(*

short summary
=================
Class provides assert statements
for 8-bit windows-1252 and UTF-16 strings with an undifined length.

.. attention:: 
	All strings are handled as null terminated byte/word streams.
	For windows-1252 is end of the string 16#00
	For UTF-16 is end of the string 16#00_00

.. attention:: 
	The interface :ref:`IAnyStringAssertions` uses ``ANY_STRING``, 
	for this it's not possible to use literals/constants,
	because for ``ANY`` types generates the compiler ``__SYSTEM.AnyType``
	and ``__SYSTEM.AnyType`` contains a pointer  

.. <legal notes>

legal notes
=================
| SPDX-FileCopyrightText: © 2022 ekvip automation GmbH <info@ekvip.de>
| SPDX-License-Identifier: Apache-2.0
| For details check: Apache-2.0_

.. _Apache-2.0: https://www.apache.org/licenses/LICENSE-2.0

.. </legal notes>

methods and properties
=======================

*)

{attribute 'reflection'}
FUNCTION_BLOCK INTERNAL AnyStringAssertions EXTENDS AbstactAssertion IMPLEMENTS IAnyStringAssertions
VAR
	(* class to handle the windows-1252 string assertions *)  
	win1252Assertions	:Windows1252StringPointerAssertions();
	(* class to handle the windows-1252 string assertions *)  
	utf16Assertions		:Utf16StringPointerAssertions();	
END_VAR

(*

short summary
=================
This abstract property returns the class name of the concrete object, 
It's for debugging purpose

.. <legal notes>

legal notes
=================
| SPDX-FileCopyrightText: © 2022 ekvip automation GmbH <info@ekvip.de>
| SPDX-License-Identifier: Apache-2.0
| For details check: Apache-2.0_

.. _Apache-2.0: https://www.apache.org/licenses/LICENSE-2.0

.. </legal notes>

*)

PROPERTY className :CNM_AbstractObject.ClassName
GET
className := 'CNM_AssertionInterfaceLib.AnyStringAssertions';
END_GET
END_PROPERTY

(*

short summary
=================
This assertion method checks if the current string ``stringToCheck`` contains the search string

.. attention:: 
	All strings are handled as null terminated byte/word streams.
	For windows-1252 is end of the string 16#00
	For UTF-16 is end of the string 16#00_00

.. attention:: 
	Method uses ``ANY_STRING`` and for this it's not possible
	to use literals/constants, because for ``ANY`` types the
	compiler generates``__SYSTEM.AnyType`` and 
	``__SYSTEM.AnyType`` contains a pointer  

.. <legal notes>

legal notes
=================
| SPDX-FileCopyrightText: © 2022 ekvip automation GmbH <info@ekvip.de>
| SPDX-License-Identifier: Apache-2.0
| For details check: Apache-2.0_

.. _Apache-2.0: https://www.apache.org/licenses/LICENSE-2.0

.. </legal notes>

parameters
=================

*)

METHOD contains
VAR_INPUT
	(* current string to check *)
	stringToCheck	:ANY_STRING;
	(* string must be found in ``stringToCheck`` *)
	searchString	:ANY_STRING;
	(* ``TRUE`` means ignore cases; ``FALSE`` means cases must be equal too *)
	ignoreCases		:BOOL;
	(* message if the assertion is false *)
	message			:AssertMessage;
END_VAR
IF (stringToCheck.TypeClass <> searchString.TypeClass) THEN
	THIS^.assertionWasWrong(message, THIS^.getDebugInfo('contains'));
	RETURN;
END_IF

IF (stringToCheck.TypeClass = __SYSTEM.TYPE_CLASS.TYPE_STRING) THEN
	THIS^.win1252Assertions.win1252Contains(
		stringToCheck := stringToCheck.pValue,
		searchString := searchString.pValue,
		ignoreCases := ignoreCases,
		message := message
	);
ELSIF (stringToCheck.TypeClass = __SYSTEM.TYPE_CLASS.TYPE_WSTRING) THEN
	THIS^.utf16Assertions.utf16Contains(
		stringToCheck := stringToCheck.pValue,
		searchString := searchString.pValue,
		ignoreCases := ignoreCases,
		message := message
	);	
END_IF
END_METHOD

(*

short summary
=================
This assertion method checks if the current string ``stringToCheck`` not contains the search string

.. attention:: 
	All strings are handled as null terminated byte/word streams.
	For windows-1252 is end of the string 16#00
	For UTF-16 is end of the string 16#00_00

.. attention:: 
	Method uses ``ANY_STRING`` and for this it's not possible
	to use literals/constants, because for ``ANY`` types the
	compiler generates``__SYSTEM.AnyType`` and 
	``__SYSTEM.AnyType`` contains a pointer  

.. <legal notes>

legal notes
=================
| SPDX-FileCopyrightText: © 2022 ekvip automation GmbH <info@ekvip.de>
| SPDX-License-Identifier: Apache-2.0
| For details check: Apache-2.0_

.. _Apache-2.0: https://www.apache.org/licenses/LICENSE-2.0

.. </legal notes>

parameters
=================

*)

METHOD containsNo
VAR_INPUT
	(* current string to check *)
	stringToCheck	:ANY_STRING;
	(* string that must not be found in ``stringToCheck`` *)
	searchString	:ANY_STRING;
	(* ``TRUE`` means ignore cases; ``FALSE`` means cases must be equal too *)
	ignoreCases		:BOOL;
	(* message if the assertion is false *)
	message			:AssertMessage;
END_VAR
IF (stringToCheck.TypeClass <> searchString.TypeClass) THEN
	THIS^.assertionWasWrong(message, THIS^.getDebugInfo('containsNo'));
	RETURN;
END_IF

IF (stringToCheck.TypeClass = __SYSTEM.TYPE_CLASS.TYPE_STRING) THEN
	THIS^.win1252Assertions.win1252ContainsNo(
		stringToCheck := stringToCheck.pValue,
		searchString := searchString.pValue,
		ignoreCases := ignoreCases,
		message := message
	);
ELSIF (stringToCheck.TypeClass = __SYSTEM.TYPE_CLASS.TYPE_WSTRING) THEN
	THIS^.utf16Assertions.utf16ContainsNo(
		stringToCheck := stringToCheck.pValue,
		searchString := searchString.pValue,
		ignoreCases := ignoreCases,
		message := message
	);
END_IF
END_METHOD

(*

short summary
=================
This assertion method checks if the current string ``stringToCheck`` ends with ``end``

.. attention:: 
	All strings are handled as null terminated byte/word streams.
	For windows-1252 is end of the string 16#00
	For UTF-16 is end of the string 16#00_00

.. attention:: 
	Method uses ``ANY_STRING`` and for this it's not possible
	to use literals/constants, because for ``ANY`` types the
	compiler generates``__SYSTEM.AnyType`` and 
	``__SYSTEM.AnyType`` contains a pointer  

.. attention:: 
	end of the string is **ALWAYS** the right side of the string 
	even for writings which written from right to left like Hebrew or Arabic

.. <legal notes>

legal notes
=================
| SPDX-FileCopyrightText: © 2022 ekvip automation GmbH <info@ekvip.de>
| SPDX-License-Identifier: Apache-2.0
| For details check: Apache-2.0_

.. _Apache-2.0: https://www.apache.org/licenses/LICENSE-2.0

.. </legal notes>

parameters
=================

*)

METHOD endsWith
VAR_INPUT
	(* current string to check *)
	stringToCheck	:ANY_STRING;
	(* expected end of ``stringToCheck`` *)
	end				:ANY_STRING;
	(* ``TRUE`` means ignore cases; ``FALSE`` means cases must be equal too *)
	ignoreCases		:BOOL;
	(* ``TRUE`` means truncation of spaces on the right side of ``stringToCheck``*)
	trim			:BOOL;
	(* message if the assertion is false *)
	message			:AssertMessage;
END_VAR
IF (stringToCheck.TypeClass <> end.TypeClass) THEN
	THIS^.assertionWasWrong(message, THIS^.getDebugInfo('endsWith'));
	RETURN;
END_IF

IF (stringToCheck.TypeClass = __SYSTEM.TYPE_CLASS.TYPE_STRING) THEN
	THIS^.win1252Assertions.win1252EndsWith(
		stringToCheck := stringToCheck.pValue,
		end := end.pValue,
		ignoreCases := ignoreCases,
		trim := trim,
		message := message
	);
ELSIF (stringToCheck.TypeClass = __SYSTEM.TYPE_CLASS.TYPE_WSTRING) THEN
	THIS^.utf16Assertions.utf16EndsWith(
		stringToCheck := stringToCheck.pValue,
		end := end.pValue,
		ignoreCases := ignoreCases,
		trim := trim,
		message := message
	);	
END_IF
END_METHOD

(*

short summary
=================
This assertion method checks if the current string ``stringToCheck`` is empty

.. attention:: 
	All strings are handled as null terminated byte/word streams.
	For windows-1252 is end of the string 16#00
	For UTF-16 is end of the string 16#00_00

.. attention:: 
	Method uses ``ANY_STRING`` and for this it's not possible
	to use literals/constants, because for ``ANY`` types the
	compiler generates``__SYSTEM.AnyType`` and 
	``__SYSTEM.AnyType`` contains a pointer  

.. <legal notes>

legal notes
=================
| SPDX-FileCopyrightText: © 2022 ekvip automation GmbH <info@ekvip.de>
| SPDX-License-Identifier: Apache-2.0
| For details check: Apache-2.0_

.. _Apache-2.0: https://www.apache.org/licenses/LICENSE-2.0

.. </legal notes>

parameters
=================

*)

METHOD isEmpty
VAR_INPUT
	(* current string to check *)
	stringToCheck	:ANY_STRING;
	(* message if the assertion is false *)
	message			:AssertMessage;
END_VAR
VAR CONSTANT
	(* strings are null terminated *)
	END_OF_WINDOWS_1252_STRING	:BYTE := 16#00;
	(* strings are null terminated *)
	END_OF_UTF16_STRING	:WORD := 16#0000;
END_VAR
IF (stringToCheck.TypeClass = __SYSTEM.TYPE_CLASS.TYPE_STRING) THEN
	IF (stringToCheck.pValue^ <> END_OF_WINDOWS_1252_STRING) THEN
		THIS^.assertionWasWrong(message, THIS^.getDebugInfo('isEmpty'));
	END_IF
ELSIF (stringToCheck.TypeClass = __SYSTEM.TYPE_CLASS.TYPE_WSTRING) THEN
	IF (stringToCheck.pValue^ <> END_OF_UTF16_STRING) THEN
		THIS^.assertionWasWrong(message, THIS^.getDebugInfo('isEmpty'));
	END_IF
END_IF
END_METHOD

(*

short summary
=================
This assertion method checks if the current string ``stringToCheck`` is equal to ``expected``

.. attention:: 
	All strings are handled as null terminated byte/word streams.
	For windows-1252 is end of the string 16#00
	For UTF-16 is end of the string 16#00_00

.. attention:: 
	Method uses ``ANY_STRING`` and for this it's not possible
	to use literals/constants, because for ``ANY`` types the
	compiler generates``__SYSTEM.AnyType`` and 
	``__SYSTEM.AnyType`` contains a pointer  

.. <legal notes>

legal notes
=================
| SPDX-FileCopyrightText: © 2022 ekvip automation GmbH <info@ekvip.de>
| SPDX-License-Identifier: Apache-2.0
| For details check: Apache-2.0_

.. _Apache-2.0: https://www.apache.org/licenses/LICENSE-2.0

.. </legal notes>

parameters
=================

*)

METHOD isEqualTo
VAR_INPUT
	(* current string to check *)
	stringToCheck	:ANY_STRING;
	(* ``stringToCheck`` must be equal to expected *)
	expected		:ANY_STRING;
	(* ``TRUE`` means ignore cases; ``FALSE`` means cases must be equal too *)
	ignoreCases		:BOOL;
	(* message if the assertion is false *)
	message			:AssertMessage;
END_VAR
IF (stringToCheck.TypeClass <> expected.TypeClass) THEN
	THIS^.assertionWasWrong(message, THIS^.getDebugInfo('isEqualTo'));
	RETURN;
END_IF

IF (stringToCheck.TypeClass = __SYSTEM.TYPE_CLASS.TYPE_STRING) THEN
	THIS^.win1252Assertions.win1252IsEqualTo(
		stringToCheck := stringToCheck.pValue,
		expected := expected.pValue,
		ignoreCases := ignoreCases,
		message := message
	);
ELSIF (stringToCheck.TypeClass = __SYSTEM.TYPE_CLASS.TYPE_WSTRING) THEN
	THIS^.utf16Assertions.utf16IsEqualTo(
		stringToCheck := stringToCheck.pValue,
		expected := expected.pValue,
		ignoreCases := ignoreCases,
		message := message
	);	
END_IF
END_METHOD

(*

short summary
=================
This assertion method checks if the current string ``stringToCheck`` is not empty

.. attention:: 
	All strings are handled as null terminated byte/word streams.
	For windows-1252 is end of the string 16#00
	For UTF-16 is end of the string 16#00_00

.. attention:: 
	Method uses ``ANY_STRING`` and for this it's not possible
	to use literals/constants, because for ``ANY`` types the
	compiler generates``__SYSTEM.AnyType`` and 
	``__SYSTEM.AnyType`` contains a pointer  

.. <legal notes>

legal notes
=================
| SPDX-FileCopyrightText: © 2022 ekvip automation GmbH <info@ekvip.de>
| SPDX-License-Identifier: Apache-2.0
| For details check: Apache-2.0_

.. _Apache-2.0: https://www.apache.org/licenses/LICENSE-2.0

.. </legal notes>

parameters
=================

*)

METHOD isNotEmpty
VAR_INPUT
	(* current string to check *)
	stringToCheck	:ANY_STRING;
	(* message if the assertion is false *)
	message			:AssertMessage;
END_VAR
VAR CONSTANT
	(* strings are null terminated *)
	END_OF_WINDOWS_1252_STRING	:BYTE := 16#00;
	(* strings are null terminated *)
	END_OF_UTF16_STRING	:WORD := 16#0000;
END_VAR
IF (stringToCheck.TypeClass = __SYSTEM.TYPE_CLASS.TYPE_STRING) THEN
	IF (stringToCheck.pValue^ = END_OF_WINDOWS_1252_STRING) THEN
		THIS^.assertionWasWrong(message, THIS^.getDebugInfo('isNotEmpty'));
	END_IF
ELSIF (stringToCheck.TypeClass = __SYSTEM.TYPE_CLASS.TYPE_WSTRING) THEN
	IF (stringToCheck.pValue^ = END_OF_UTF16_STRING) THEN
		THIS^.assertionWasWrong(message, THIS^.getDebugInfo('isNotEmpty'));
	END_IF
END_IF
END_METHOD

(*

short summary
=================
This assertion method checks if the current string ``stringToCheck`` is not equal to ``unexpected``

.. attention:: 
	All strings are handled as null terminated byte/word streams.
	For windows-1252 is end of the string 16#00
	For UTF-16 is end of the string 16#00_00

.. attention:: 
	Method uses ``ANY_STRING`` and for this it's not possible
	to use literals/constants, because for ``ANY`` types the
	compiler generates``__SYSTEM.AnyType`` and 
	``__SYSTEM.AnyType`` contains a pointer  

.. <legal notes>

legal notes
=================
| SPDX-FileCopyrightText: © 2022 ekvip automation GmbH <info@ekvip.de>
| SPDX-License-Identifier: Apache-2.0
| For details check: Apache-2.0_

.. _Apache-2.0: https://www.apache.org/licenses/LICENSE-2.0

.. </legal notes>

parameters
=================

*)

METHOD isNotEqualTo
VAR_INPUT
	(* current string to check *)
	stringToCheck	:ANY_STRING;
	(* ``stringToCheck`` must be not equal to expected *)
	unexpected		:ANY_STRING;
	(* ``TRUE`` means ignore cases; ``FALSE`` means cases must be equal too *)
	ignoreCases		:BOOL;
	(* message if the assertion is false *)
	message			:AssertMessage;
END_VAR
IF (stringToCheck.TypeClass <> unexpected.TypeClass) THEN
	RETURN;
END_IF

IF (stringToCheck.TypeClass = __SYSTEM.TYPE_CLASS.TYPE_STRING) THEN
	THIS^.win1252Assertions.win1252IsNotEqualTo(
		stringToCheck := stringToCheck.pValue,
		unexpected := unexpected.pValue,
		ignoreCases := ignoreCases,
		message := message
	);
ELSIF (stringToCheck.TypeClass = __SYSTEM.TYPE_CLASS.TYPE_WSTRING) THEN
	THIS^.utf16Assertions.utf16IsNotEqualTo(
		stringToCheck := stringToCheck.pValue,
		unexpected := unexpected.pValue,
		ignoreCases := ignoreCases,
		message := message
	);	
END_IF
END_METHOD

(*

short summary
=================
This assertion method checks if the current string ``stringToCheck`` is length
is between ``minLenght`` and ``maxLenght``

.. attention:: 
	All strings are handled as null terminated byte/word streams.
	For windows-1252 is end of the string 16#00
	For UTF-16 is end of the string 16#00_00

.. attention:: 
	Method uses ``ANY_STRING`` and for this it's not possible
	to use literals/constants, because for ``ANY`` types the
	compiler generates``__SYSTEM.AnyType`` and 
	``__SYSTEM.AnyType`` contains a pointer  

.. <legal notes>

legal notes
=================
| SPDX-FileCopyrightText: © 2022 ekvip automation GmbH <info@ekvip.de>
| SPDX-License-Identifier: Apache-2.0
| For details check: Apache-2.0_

.. _Apache-2.0: https://www.apache.org/licenses/LICENSE-2.0

.. </legal notes>

parameters
=================

*)

METHOD lenghtIsBetween
VAR_INPUT
	(* current string to check *)
	stringToCheck	:ANY_STRING;
	(* lower limit of the string length *)
	minLenght		:UDINT;
	(* upper limit of the string length *)
	maxLenght		:UDINT;
	(* message if the assertion is false *)
	message			:AssertMessage;
END_VAR
IF (stringToCheck.TypeClass = __SYSTEM.TYPE_CLASS.TYPE_STRING) THEN
	THIS^.win1252Assertions.win1252LengthIsBetween(
		stringToCheck	:= stringToCheck.pValue,
		minLenght		:= minLenght,
		maxLenght		:= maxLenght,
		message			:= message
	);
ELSIF (stringToCheck.TypeClass = __SYSTEM.TYPE_CLASS.TYPE_WSTRING) THEN
	THIS^.utf16Assertions.utf16LengthIsBetween(
		stringToCheck	:= stringToCheck.pValue,
		minLenght		:= minLenght,
		maxLenght		:= maxLenght,
		message			:= message
	);	
END_IF
END_METHOD

(*

short summary
=================
This assertion method checks if the current string ``stringToCheck`` is length
is equal to ``expectedLength``

.. attention:: 
	All strings are handled as null terminated byte/word streams.
	For windows-1252 is end of the string 16#00
	For UTF-16 is end of the string 16#00_00

.. attention:: 
	Method uses ``ANY_STRING`` and for this it's not possible
	to use literals/constants, because for ``ANY`` types the
	compiler generates``__SYSTEM.AnyType`` and 
	``__SYSTEM.AnyType`` contains a pointer  

.. <legal notes>

legal notes
=================
| SPDX-FileCopyrightText: © 2022 ekvip automation GmbH <info@ekvip.de>
| SPDX-License-Identifier: Apache-2.0
| For details check: Apache-2.0_

.. _Apache-2.0: https://www.apache.org/licenses/LICENSE-2.0

.. </legal notes>

parameters
=================

*)

METHOD lenghtIsExact
VAR_INPUT
	(* current string to check *)
	stringToCheck	:ANY_STRING;
	(* expected length of ``stringToCheck`` *)
	expectedLength	:UDINT;
	(* message if the assertion is false *)
	message			:AssertMessage;
END_VAR
IF (stringToCheck.TypeClass = __SYSTEM.TYPE_CLASS.TYPE_STRING) THEN
	THIS^.win1252Assertions.win1252LenghtIsExact(
		stringToCheck	:= stringToCheck.pValue,
		expectedLength	:= expectedLength,
		message			:= message
	);
ELSIF (stringToCheck.TypeClass = __SYSTEM.TYPE_CLASS.TYPE_WSTRING) THEN
	THIS^.utf16Assertions.utf16LenghtIsExact(
		stringToCheck	:= stringToCheck.pValue,
		expectedLength	:= expectedLength,
		message			:= message
	);	
END_IF
END_METHOD

(*

short summary
=================
This assertion method checks if the current string ``stringToCheck`` is length
is equal or less than to ``maxLength``

.. attention:: 
	All strings are handled as null terminated byte/word streams.
	For windows-1252 is end of the string 16#00
	For UTF-16 is end of the string 16#00_00

.. attention:: 
	Method uses ``ANY_STRING`` and for this it's not possible
	to use literals/constants, because for ``ANY`` types the
	compiler generates``__SYSTEM.AnyType`` and 
	``__SYSTEM.AnyType`` contains a pointer  

.. <legal notes>

legal notes
=================
| SPDX-FileCopyrightText: © 2022 ekvip automation GmbH <info@ekvip.de>
| SPDX-License-Identifier: Apache-2.0
| For details check: Apache-2.0_

.. _Apache-2.0: https://www.apache.org/licenses/LICENSE-2.0

.. </legal notes>

parameters
=================

*)

METHOD lenghtIsMax
VAR_INPUT
	(* current string to check *)
	stringToCheck	:ANY_STRING;
	(* upper limit of the length of ``stringToCheck`` *)
	maxLength		:UDINT;
	(* message if the assertion is false *)
	message			:AssertMessage;
END_VAR
IF (stringToCheck.TypeClass = __SYSTEM.TYPE_CLASS.TYPE_STRING) THEN
	THIS^.win1252Assertions.win1252LenghtIsMax(
		stringToCheck	:= stringToCheck.pValue,
		maxLength		:= maxLength,
		message			:= message
	);
ELSIF (stringToCheck.TypeClass = __SYSTEM.TYPE_CLASS.TYPE_WSTRING) THEN
	THIS^.utf16Assertions.utf16LenghtIsMax(
		stringToCheck	:= stringToCheck.pValue,
		maxLength		:= maxLength,
		message			:= message
	);	
END_IF
END_METHOD

(*

short summary
=================
This assertion method checks if the current string ``stringToCheck`` is length
is equal or grater than to ``minLength``

.. attention:: 
	All strings are handled as null terminated byte/word streams.
	For windows-1252 is end of the string 16#00
	For UTF-16 is end of the string 16#00_00

.. attention:: 
	Method uses ``ANY_STRING`` and for this it's not possible
	to use literals/constants, because for ``ANY`` types the
	compiler generates``__SYSTEM.AnyType`` and 
	``__SYSTEM.AnyType`` contains a pointer  

.. <legal notes>

legal notes
=================
| SPDX-FileCopyrightText: © 2022 ekvip automation GmbH <info@ekvip.de>
| SPDX-License-Identifier: Apache-2.0
| For details check: Apache-2.0_

.. _Apache-2.0: https://www.apache.org/licenses/LICENSE-2.0

.. </legal notes>

parameters
=================

*)

METHOD lenghtIsMin
VAR_INPUT
	(* current string to check *)
	stringToCheck	:ANY_STRING;
	(* lower limit of the length of ``stringToCheck`` *)
	minLength		:UDINT;
	(* message if the assertion is false *)
	message			:AssertMessage;
END_VAR
IF (stringToCheck.TypeClass = __SYSTEM.TYPE_CLASS.TYPE_STRING) THEN
	THIS^.win1252Assertions.win1252LenghtIsMin(
		stringToCheck	:= stringToCheck.pValue,
		minLength		:= minLength,
		message			:= message
	);
ELSIF (stringToCheck.TypeClass = __SYSTEM.TYPE_CLASS.TYPE_WSTRING) THEN
	THIS^.utf16Assertions.utf16LenghtIsMin(
		stringToCheck	:= stringToCheck.pValue,
		minLength		:= minLength,
		message			:= message
	);
END_IF
END_METHOD

(*

short summary
=================
This methods is the setter for the callback class if an assertion was false

.. <legal notes>

legal notes
=================
| SPDX-FileCopyrightText: © 2022 ekvip automation GmbH <info@ekvip.de>
| SPDX-License-Identifier: Apache-2.0
| For details check: Apache-2.0_

.. _Apache-2.0: https://www.apache.org/licenses/LICENSE-2.0

.. </legal notes>

parameters
=================

*)

METHOD setCallBack
VAR_INPUT
	(* the class that must be informed if an assertion is false *)
	callBack	:IAssertCallback;  
END_VAR
SUPER^.setCallBack(callBack);
THIS^.win1252Assertions.setCallBack(callBack);
THIS^.utf16Assertions.setCallBack(callBack);
END_METHOD

(*

short summary
=================
This assertion method checks if the current string ``stringToCheck`` starts with ``start``

.. attention:: 
	All strings are handled as null terminated byte/word streams.
	For windows-1252 is end of the string 16#00
	For UTF-16 is end of the string 16#00_00

.. attention:: 
	Method uses ``ANY_STRING`` and for this it's not possible
	to use literals/constants, because for ``ANY`` types the
	compiler generates``__SYSTEM.AnyType`` and 
	``__SYSTEM.AnyType`` contains a pointer  

.. attention:: 
	start of the string is **ALWAYS** the left side of the string 
	even for writings which written from right to left like Hebrew or Arabic

.. <legal notes>

legal notes
=================
| SPDX-FileCopyrightText: © 2022 ekvip automation GmbH <info@ekvip.de>
| SPDX-License-Identifier: Apache-2.0
| For details check: Apache-2.0_

.. _Apache-2.0: https://www.apache.org/licenses/LICENSE-2.0

.. </legal notes>

parameters
=================

*)

METHOD startsWith
VAR_INPUT
	(* current string to check *)
	stringToCheck	:ANY_STRING;
	(* expected start of ``stringToCheck`` *)
	start			:ANY_STRING;
	(* ``TRUE`` means ignore cases; ``FALSE`` means cases must be equal too *)
	ignoreCases		:BOOL;
	(* ``TRUE`` means truncation of spaces on the left side of ``stringToCheck``*)
	trim			:BOOL;
	(* message if the assertion is false *)
	message			:AssertMessage;
END_VAR
IF (stringToCheck.TypeClass <> start.TypeClass) THEN
	THIS^.assertionWasWrong(message, THIS^.getDebugInfo('startsWith'));
	RETURN;
END_IF

IF (stringToCheck.TypeClass = __SYSTEM.TYPE_CLASS.TYPE_STRING) THEN
	THIS^.win1252Assertions.win1252StartsWith(
		stringToCheck := stringToCheck.pValue,
		start := start.pValue,
		ignoreCases := ignoreCases,
		trim := trim,
		message := message
	);
ELSIF (stringToCheck.TypeClass = __SYSTEM.TYPE_CLASS.TYPE_WSTRING) THEN
	THIS^.utf16Assertions.utf16StartsWith(
		stringToCheck := stringToCheck.pValue,
		start := start.pValue,
		ignoreCases := ignoreCases,
		trim := trim,
		message := message
	);
END_IF
END_METHOD

END_FUNCTION_BLOCK

(* stored: Version 1.1.0.1, ProductVersion 3.1.4024.12
   POU AnyStringAssertions: Id {fb248394-cb20-4e0b-96e4-b40ac93ae790}, SpecialFunc None
   Property className: Id {fcc2d213-734a-4988-a56c-58e116884246}
   Get Get: Id {65e2fc47-ed60-4e11-b462-d54a00eb1b07}
   Method contains: Id {bf0ab0d6-fe3a-4edc-a46b-d453067bd3cc}
   Method containsNo: Id {8225714f-42b0-45a3-bb95-a08686884681}
   Method endsWith: Id {2caa6531-5c1e-4058-bb14-79e815fd424d}
   Method isEmpty: Id {200f5764-869a-419f-9fc7-791ed622a0f2}
   Method isEqualTo: Id {d4d26bf4-0744-4ca1-8927-f44aea35a280}
   Method isNotEmpty: Id {835874ca-5f9b-4d9b-b2b8-1067b6d4b0ec}
   Method isNotEqualTo: Id {559d8201-64ec-4b0d-8552-16733b596597}
   Method lenghtIsBetween: Id {85ae0d0b-fcee-4e49-a9cb-1428d7808523}
   Method lenghtIsExact: Id {86be1f58-2b02-4c78-b0cb-0df1dfc206a7}
   Method lenghtIsMax: Id {aaf05057-5f7a-4682-9d17-e178e35c37eb}
   Method lenghtIsMin: Id {db33c3ef-31df-4fde-a320-0a6fd13a6db6}
   Method setCallBack: Id {e8e733fa-1cf4-4c00-a65d-918e41c02968}
   Method startsWith: Id {11d9b96d-e584-4359-aa8c-6388497efbf5} *)
